// Generated by tiagen - edit the machine spec, not this file.
ORGANIZATION_BLOCK "Main"
TITLE = 'Program cycle'
{ S7_Optimized_Access := 'TRUE' }
VERSION : 0.1
BEGIN
    "DB_TransferStation"();
END_ORGANIZATION_BLOCK

(*
   Calls the machine FB through its instance DB DB_TransferStation.

   The build plan deletes the project's default Main [OB1] before importing
   this one, so that OB1 ends up as this SCL block. If your TIA version
   refuses the import, keep the original Main [OB1] and add the single line
   DB_TransferStation(); to it by hand - that is the only manual code step.
*)
